// TwinCAT 3 PLC project Example_1
// ProgramVersion: 3.1.4024.0
// libraries:
//   Tc2_Standard, * (Beckhoff Automation GmbH)
//   Tc2_System, * (Beckhoff Automation GmbH)
//   Tc2_Utilities, * (Beckhoff Automation GmbH)
//   Tc3_Module, * (Beckhoff Automation GmbH)
// project tree:
//   DUTs/ ST_Point.TcDUT
//   GVLs/ GVL_Var.TcGVL
//   / PlcTask.TcTTO
//   POUs/ FB_PumpController.TcPOU, FB_SimulatedIO.TcPOU, KukaRobot.TcPOU, MAIN.TcPOU, FB_Pump.TcPOU
// real-time tasks:
//   TASK PlcTask: cycle T#10ms, priority 20, ADS port 350
// I/O:
//   DEVICE Device 1 (EtherCAT) (disabled), AmsNetId 172.24.64.1.2.1
//     Term 1 (EK1100) [EK1100 EtherCAT Coupler (2A E-Bus)]
//       Term 2 (EL3024) [EL3024 4Ch. Ana. Input 4-20mA DIFF]
//       Term 3 (EL2634) [EL2634 4Ch. Relay Output, NO (250V AC / 30V DC)]
//     Box 4 (KRC4 secondary EL6695-1001) [KRC4 secondary EL6695-1001]
//       modules: Module 1 (Sync Inputs), Module 2 (Safety Data Bitf  (8 Byte)), Module 3 (Default IO)
// variable links:
//   Example_1/Example_1 Instance <-> Device 1 (EtherCAT)/Box 4 (KRC4 secondary EL6695-1001)
//     PlcTask Outputs/MAIN.KukaBot.wOutputWord <-> Module 3 (Default IO)/Std. Out (4 Bytes)/Output DWORD 0

CONFIGURATION Example_1
    RESOURCE PLC ON TwinCAT3
        TASK PlcTask(INTERVAL := T#10ms, PRIORITY := 20);
        PROGRAM MAIN WITH PlcTask : MAIN;
    END_RESOURCE
END_CONFIGURATION

// ---- DUTs/ST_Point.TcDUT
TYPE ST_Point :
	STRUCT
		x : INT;
		y : REAL;
	END_STRUCT
END_TYPE

// ---- GVLs/GVL_Var.TcGVL
{attribute 'qualified_only'}
VAR_GLOBAL
END_VAR
VAR_GLOBAL
	// Pressure within the pumps
	nPressure: REAL := 1;
	// Whether the pump is on
	bPump: BOOL := FALSE;
	bValve : BOOL := FALSE;
	bLeakDetected : BOOL := FALSE;
	bBrokenPump : BOOL := FALSE;
	bControllerError : BOOL := FALSE;
	bReset: BOOL := FALSE;
	nPumpGain : LREAL := 0.01;
	nPassiveLoss : LREAL := 0.001;
	nValveLoss : LREAL := 0.02;
	nKp : LREAL := 0.001;
	nTn : LREAL := 0.1;
	nTv : LREAL := 0.1;
	nTd : LREAL := 0.1;
END_VAR

// ---- POUs/MAIN.TcPOU
PROGRAM MAIN
VAR
	// Objects
	SimulatedIO : FB_SimulatedIO;
	Pump : FB_Pump;
	PumpController : FB_PumpController := (nTargetPressure := TARGET_PRESSURE, nMaximumPressure := MAXIMUM_PRESSURE,
		nMinimumPressure := MINIMUM_PRESSURE, nInitialPressure := Pump.nPressure);
	KukaBot : KukaRobot;
	
	// Variables for Graph
	aGraphPoints : ARRAY[1..1, 1..1000] OF ST_Point;
	nPollDelay : UINT := 10; 
	nCurrentPoint : INT := 1;
	nPollCount : UINT := 0;
	
	// HMI Variables
	bTurnPumpControllerOn : BOOL := FALSE;
	bEmergencyStopPump : BOOL := FALSE;
	sState : STRING(20) := 'IDLE';
	bManualPump : BOOL := FALSE;
	bManualRelease : BOOL := FALSE;
	
	// Main Loop Variables
	bPumpState : BOOL := FALSE;
	bValveState : BOOL := FALSE;
END_VAR

VAR CONSTANT
	MAXIMUM_PRESSURE : USINT := 10;
	MINIMUM_PRESSURE : USINT := 8;
	TARGET_PRESSURE : USINT := 9;
END_VAR

IF GVL_VAR.bReset THEN // RESET State
	bEmergencyStopPump := FALSE;
	GVL_VAR.bBrokenPump := FALSE;
	GVL_Var.bLeakDetected := FALSE;
	GVL_VAR.bControllerError := FALSE;
	bTurnPumpControllerOn := FALSE;
	PumpController.Reset();
	bManualPump := FALSE;
	bManualRelease := FALSE;
	GVL_VAR.bReset := FALSE;
	
ELSIF GVL_VAR.bBrokenPump THEN // Something Broken State
	sState := 'SMT_BROKE';
	Shutdown();
	
ELSIF bEmergencyStopPump THEN // Emergency Stopped State
	sState := 'E_STOPPED';
	Shutdown();
	
ELSIF GVL_Var.bLeakDetected THEN // Leak Detected State
	sState := 'LEAK!';
	Shutdown();
	
ELSIF GVL_Var.bControllerError THEN // Leak Detected State
	sState := 'CtrlErr!';
	Shutdown();
	
ELSE // All Systems Normal
	sState := 'IDLING';
	IF bTurnPumpControllerOn THEN
		// PumpController.RunSimpleController(bTurnPumpControllerOn); // Simple Controller
		PumpController.RunPIDController(bTurnPumpControllerOn); // PID Controller
		bPumpState := PumpController.bPumpState;
		bValveState := PumpController.bValveState;
		Pump.SetRelay(bPumpState);
		Pump.SetValve(bValveState);
		IF bPumpState THEN
			sState := 'PUMPING';
		ELSIF bValveState THEN
			sState := 'RELEASING';
		END_IF
	ELSIF bManualRelease THEN
		sState := 'M_RELEASE';
		GVL_VAR.nValveLoss := 0.02;
		Pump.SetValve(TRUE);
		Pump.SetRelay(FALSE);
	ELSIF bManualPump THEN
		sState := 'M_PUMPING';
		GVL_VAR.nPumpGain := 0.01;
		Pump.SetRelay(TRUE);
		Pump.SetValve(FALSE);
	ELSE
		PUMP.SetRelay(FALSE);
		PUMP.SetValve(FALSE);
	END_IF
END_IF

// Save pressure data for graph
IF nCurrentPoint > 1000 THEN
	nCurrentPoint := 2;
	nPollCount := 2;
ELSIF nPollCount > 9 THEN
	aGraphPoints[1, nCurrentPoint].x := nCurrentPoint;
	aGraphPoints[1, nCurrentPoint].y := Pump.nPressure;
	nPollCount := 0;
	nCurrentPoint := 1 + nCurrentPoint;
ELSE
	nPollCount := nPollCount + 1;
END_IF

KukaBot.SendData(GVL_Var.bLeakDetected);
// Simulate I/O
SimulatedIO();
Pump(); // Simulated Pump output

METHOD Shutdown : BOOL
Pump.SetRelay(FALSE);
bTurnPumpControllerOn := FALSE;
Shutdown := TRUE;
END_METHOD

END_PROGRAM

// ---- POUs/FB_SimulatedIO.TcPOU
FUNCTION_BLOCK FB_SimulatedIO

IF GVL_VAR.bPump THEN
	GVL_VAR.nPressure := GVL_VAR.nPressure + GVL_VAR.nPumpGain;
ELSIF GVL_VAR.nPressure > 1 THEN
	IF GVL_VAR.bValve THEN
		GVL_VAR.nPressure := GVL_VAR.nPressure - GVL_VAR.nValveLoss;
	ELSE
		GVL_VAR.nPressure := GVL_VAR.nPressure - GVL_VAR.nPassiveLoss;	
	END_IF
ELSE
	GVL_VAR.nPressure := 1;
END_IF

END_FUNCTION_BLOCK

// ---- POUs/FB_Pump.TcPOU
FUNCTION_BLOCK FB_Pump
VAR_OUTPUT
	nPressure: REAL; // [Volts]
END_VAR
VAR
	// bRelayOn AT %Q* : BOOL := FALSE; // True = On
	bRelayOn : BOOL := FALSE;
	// nCurrentPressure AT %I* : REAL; // Volts
	bValveOpen : BOOL := FALSE;
END_VAR

// For Simulation
IF bValveOpen THEN
	GVL_VAR.bValve := TRUE;
	GVL_VAR.bPump := FALSE;
ELSIF bRelayOn THEN
	GVL_VAR.bPump := TRUE;
	GVL_VAR.bValve := FALSE;
ELSE
	GVL_VAR.bPump := FALSE;
	GVL_VAR.bValve := FALSE;
END_IF
nPressure := GVL_VAR.nPressure;

METHOD PUBLIC SetRelay : BOOL
VAR_INPUT
	bRelayState : BOOL;
END_VAR
bRelayOn := bRelayState;
SetRelay := TRUE;
END_METHOD

METHOD PUBLIC SetValve : BOOL
VAR_INPUT
	bValveState : BOOL;
END_VAR
bValveOpen := bValveState;
SetValve := TRUE;
END_METHOD

END_FUNCTION_BLOCK

// ---- POUs/FB_PumpController.TcPOU
FUNCTION_BLOCK FB_PumpController
VAR_INPUT
	nInitialTargetPressure : REAL := 9; // Volts
	nMaximumPressure : REAL := 10;
	nMinimumPressure : REAL := 8;
	nInitialPressure : REAL;
END_VAR
VAR_OUTPUT
	bPumpState : BOOL := FALSE;
	bValveState : BOOL := FALSE;
END_VAR
VAR
	// For simple pump controller
	nPumpHysteresis : REAL := 0.25;
	
	// For PID controller
	nTargetPressure : REAL := nInitialTargetPressure;
	fbPID : FB_BasicPID := (fSetpointValue := nTargetPressure, fActualValue := nInitialPressure,
fCtrlCycleTime:=0.01, fKp := GVL_VAR.nKp, fTn := GVL_VAR.nTn, fTv := GVL_VAR.nTv, fTd:= GVL_VAR.nTd);	

	// Leak detection
	nLeakHysteresis : REAL := 0.1;
	nLeakPrevPressure : REAL := nInitialPressure;
	bCheckedForLeak : BOOL := FALSE;
	
	// After <nPumpPollDelay> consecutive increases from pump, check if it's 
	// increased by at least <nPumpBrokenHysteresis>,
	nBrokenPumpHysteresis : REAL := 0.5;
	nPrevPressure : REAL := nInitialPressure;
	nPumpPollDelay : UINT := 50;
	nPollCount : UINT := 0;
END_VAR
VAR CONSTANT
	
END_VAR

METHOD PRIVATE LeakDetection : BOOL
VAR
	nPressureDiff : REAL;
END_VAR
IF bCheckedForLeak THEN
	nPressureDiff := nPrevPressure - GVL_VAR.nPressure; // Should be < 0
	nPollCount := nPollCount + 1;
	IF nPressureDiff > nBrokenPumpHysteresis THEN // Check if pump broke
		GVL_VAR.bBrokenPump := TRUE;
	ELSIF nPollCount > nPumpPollDelay THEN // Check for leak
		nPressureDiff := GVL_VAR.nPressure - nLeakPrevPressure;
		IF nPressureDiff < nLeakHysteresis THEN
			GVL_VAR.bLeakDetected := TRUE;
		END_IF
		nLeakPrevPressure := GVL_VAR.nPressure;
		nPollCount := 0;
	ELSE
		GVL_VAR.bLeakDetected := FALSE;
	END_IF
	nPrevPressure := GVL_VAR.nPressure;
	
ELSE // If it's the first call, save current pressure as prevPressure
	nPrevPressure := GVL_VAR.nPressure;
	nLeakPrevPressure := GVL_VAR.nPressure;
	bCheckedForLeak := TRUE;
	nPollCount := 1;
END_IF
END_METHOD

METHOD PUBLIC Reset : BOOL
VAR_INPUT
END_VAR
fbPID.bReset := TRUE;
bValveState := FALSE;
bPumpState := FALSE;
GVL_VAR.bLeakDetected := FALSE;
GVL_VAR.bBrokenPump := FALSE;
GVL_VAR.nPumpGain := 0.01;
GVL_VAR.nPassiveLoss := 0.001;
GVL_VAR.nValveLoss := 0.02;
Reset := TRUE; // Return val
END_METHOD

METHOD ResetLeakCheck : BOOL
bCheckedForLeak := FALSE;
nPollCount := 0;
ResetLeakCheck := TRUE;
END_METHOD

METHOD RunPIDController : BOOL
VAR_INPUT
	bState : BOOL;
END_VAR
VAR CONSTANT
	pumpGainMax : REAL := 0.5;
	pumpGainMin : LREAL := 0.001;	
	valveLossMax : REAL := 0.5;
	valveLossMin : LREAL := 0.001;
	forwardBias : REAL := 0.8;
	backBias : REAL := 1.2;
END_VAR
fbPID.fActualValue := GVL_VAR.nPressure;
fbPID();
fbPID.bReset := FALSE;

IF fbPID.nErrorStatus > 0 THEN
	bPumpState := FALSE;
	bValveState := FALSE;
	RunPIDController := FALSE;
	GVL_VAR.bControllerError := TRUE;
ELSIF GVL_VAR.nPressure > nTargetPressure THEN // Increase pressure
	bPumpState := FALSE;
	bValveState := TRUE;
	IF GVL_VAR.nPumpGain > pumpGainMin THEN
		IF fbPID.fCtrlOutput > 0 THEN // Prevents error
			GVL_VAR.nPumpGain := GVL_VAR.nPumpGain - fbPID.fCtrlOutput*backBias;
		ELSE
			GVL_VAR.nPumpGain := GVL_VAR.nPumpGain + fbPID.fCtrlOutput*backBias;
		END_IF
	ELSE
		GVL_VAR.nPumpGain := pumpGainMin;
	END_IF
	IF GVL_VAR.nValveLoss < valveLossMax THEN
		IF fbPID.fCtrlOutput > 0 THEN // Prevents error
			GVL_VAR.nValveLoss := GVL_VAR.nValveLoss + fbPID.fCtrlOutput*forwardBias;
		ELSE
			GVL_VAR.nValveLoss := GVL_VAR.nValveLoss - fbPID.fCtrlOutput*forwardBias;
		END_IF
	ELSE
		GVL_VAR.nValveLoss := valveLossMax;
	END_IF
ELSE // Decrease pressure
	bPumpState := TRUE;
	bValveState := FALSE;
	IF GVL_VAR.nValveLoss > valveLossMin THEN
		IF fbPID.fCtrlOutput > 0 THEN
			GVL_VAR.nValveLoss := GVL_VAR.nValveLoss - fbPID.fCtrlOutput*backBias;
		ELSE
			GVL_VAR.nValveLoss := GVL_VAR.nValveLoss + fbPID.fCtrlOutput*backBias;
		END_IF
	ELSE
		GVL_VAR.nValveLoss := valveLossMin;
	END_IF
	IF GVL_VAR.nPumpGain < pumpGainMax THEN
		IF fbPID.fCtrlOutput > 0 THEN
			GVL_VAR.nPumpGain := GVL_VAR.nPumpGain + fbPID.fCtrlOutput*forwardBias;
		ELSE
			GVL_VAR.nPumpGain := GVL_VAR.nPumpGain - fbPID.fCtrlOutput*forwardBias;
		END_IF
		
	ELSE
		GVL_VAR.nPumpGain := pumpGainMax;
	END_IF
END_IF
END_METHOD

METHOD RunSimpleController
VAR_INPUT
	bState : BOOL;
END_VAR
bValveState := FALSE;
IF bState THEN
	IF GVL_VAR.nPressure < nTargetPressure-nPumpHysteresis OR GVL_VAR.nPressure < nMinimumPressure+nPumpHysteresis THEN
		bPumpState := TRUE;
		LeakDetection();
	ELSIF GVL_VAR.nPressure > nTargetPressure+nPumpHysteresis OR GVL_VAR.nPressure > nMaximumPressure-nPumpHysteresis THEN
		bPumpState := FALSE;
		ResetLeakCheck();
	END_IF
ELSE
	bPumpState := FALSE;
	ResetLeakCheck();
END_IF
END_METHOD

METHOD SetTarget : BOOL
VAR_INPUT
	nNewTargetPressure : REAL;
END_VAR
nTargetPressure := nNewTargetPressure;
fbPID.fSetpointValue := nNewTargetPressure;
SetTarget := TRUE;
END_METHOD

END_FUNCTION_BLOCK

// ---- POUs/KukaRobot.TcPOU
FUNCTION_BLOCK KukaRobot
VAR_INPUT
END_VAR
VAR
	wSendData : DWORD;
END_VAR
VAR_OUTPUT
	wOutputWord AT %Q* : DWORD;
END_VAR

METHOD SendData : BOOL
VAR_INPUT
	bFailure : BOOL := FALSE;
END_VAR
IF bFailure THEN
	wOutputWord := 16#00000001;
ELSE
	wOutputWord:= 16#00000000;
END_IF
END_METHOD

END_FUNCTION_BLOCK
